ACTION ACT_Build_Ui_Strings:
                      (*
	Send to UI:	First line of Alarms
				First line of Warning
				Stop reason
*)
//PackTag.hevsPackAlarm_UI.uiTextAlarmOne := 'Complete with first Alarm';
BuildUiString := DINT_TO_STRING(PackTag.Admin.Alarm[0].ID);
BuildUiString := CONCAT(BuildUiString, ' ');
BuildUiString := CONCAT(BuildUiString, PackTag.Admin.Alarm[0].Message);
BuildUiString := CONCAT(BuildUiString, ' ');
BuildUiString := CONCAT(BuildUiString, DINT_TO_STRING(PackTag.Admin.Alarm[0].Category));
BuildUiString := CONCAT(BuildUiString, ' ');
BuildUiString := CONCAT(BuildUiString, DT_TO_STRING(PackTag.Admin.Alarm[0].DateTime));
PackTag.hevsPackAlarm_UI.uiTextAlarmOne := BuildUiString; 


BuildUiString := DINT_TO_STRING(PackTag.Admin.Warning[0].ID);
BuildUiString := CONCAT(BuildUiString, ' ');
BuildUiString := CONCAT(BuildUiString, PackTag.Admin.Warning[0].Message);
BuildUiString := CONCAT(BuildUiString, ' ');
BuildUiString := CONCAT(BuildUiString, DINT_TO_STRING(PackTag.Admin.Warning[0].Category));
BuildUiString := CONCAT(BuildUiString, ' ');
BuildUiString := CONCAT(BuildUiString, DT_TO_STRING(PackTag.Admin.Warning[0].DateTime));
PackTag.hevsPackAlarm_UI.uiTextWarningOne := BuildUiString;

BuildUiString := DINT_TO_STRING(PackTag.Admin.StopReason.ID);
BuildUiString := CONCAT(BuildUiString, ' ');
BuildUiString := CONCAT(BuildUiString, PackTag.Admin.StopReason.Message);
BuildUiString := CONCAT(BuildUiString, ' ');
BuildUiString := CONCAT(BuildUiString, DINT_TO_STRING(PackTag.Admin.StopReason.Category));
BuildUiString := CONCAT(BuildUiString, ' ');
BuildUiString := CONCAT(BuildUiString, DT_TO_STRING(PackTag.Admin.StopReason.DateTime));
PackTag.hevsPackAlarm_UI.uiTextStopReason := BuildUiString;


                    
END_ACTION
END_PROGRAM

(* www.hevs.ch Institut Systemes Industriels Project: HEVS Pack 2022 Author: Cedric Lenoir Date: 2024 August 30 This Function Block compute time statistics *)
FUNCTION_BLOCK FB_PackStatistic
  VAR_INPUT
    Enable : BOOL;
  END_VAR
  VAR_IN_OUT
    plcCurrentTime_s : UDINT;  (* E.g from PackTag.hevsPackTime.Local_date_time_seconds *)
    unitCurrentMode : E_PackModes;
    unitCurrentState : E_PackState;
    unitAdmin : HEVS_PackTag_Admin;
  END_VAR
  VAR_OUTPUT
    Active : BOOL;
  END_VAR
  VAR
    trigModeTimeCurrent : R_TRIG;  (* Detext State / Mode change *)
    trigStateTimeCurrent : R_TRIG;
    memCurrentMode : E_PackModes := E_PackModes.Invalid;
    memCurrentState : E_PackState := E_PackState.eUndefined;
    timeModeAtTrigger_s : UDINT;  (* Start time at trigger to compute current *)
    timeStateAtTrigger_s : UDINT;
    bProgramStarted : BOOL;
    timeProgramStarted_s : UDINT;
    getMemCumTimeMode : DINT;  (* Get Time In CumulativeTime for Mode and or state *)
    getMemCumTimeModeState : DINT;
  END_VAR

                  IF Enable THEN
	trigModeTimeCurrent(clk := (unitCurrentMode <> memCurrentMode));
	trigStateTimeCurrent(clk := (unitCurrentState <> memCurrentState));
	
	IF trigModeTimeCurrent.Q THEN
		timeModeAtTrigger_s := plcCurrentTime_s;
		memCurrentMode := unitCurrentMode;
		// Get Stored value to compute new cummulative time.
		getMemCumTimeMode := unitAdmin.CumulativeTime[0].ModeStateTimes[unitCurrentMode].Mode;
	END_IF
	
	IF trigStateTimeCurrent.Q THEN
		timeStateAtTrigger_s := plcCurrentTime_s;
		memCurrentState := unitCurrentState;
	END_IF
	
	// If mode or state changed
	IF trigModeTimeCurrent.Q  OR
	   trigStateTimeCurrent.Q THEN
	   getMemCumTimeModeState := unitAdmin.CumulativeTime[0].ModeStateTimes[unitCurrentMode].State[memCurrentState];
	END_IF
	
	IF NOT bProgramStarted THEN
		bProgramStarted := TRUE;
		timeProgramStarted_s := plcCurrentTime_s;
	END_IF
	
	unitAdmin.ModeTimeCurrent := UDINT_TO_DINT(plcCurrentTime_s - timeModeAtTrigger_s);
	
	unitAdmin.StateTimeCurrent := UDINT_TO_DINT(plcCurrentTime_s - timeStateAtTrigger_s);
	
	// Default for [*] time from start program
	// No retain, that is number of Sec since last restart.
	unitAdmin.CumulativeTime[0].AccTimeSinceReset := UDINT_TO_DINT(plcCurrentTime_s - timeProgramStarted_s);
	
	// Minimum protection in case of unitCurrentMode exceed 
	//	HEVS_PackTag_GVL.C_MAXMODSTATESTIMES
	IF unitCurrentMode <= HEVS_PackTag_GVL.C_MAXMODSTATESTIMES THEN
		// getMemCumTimeMode is set only at trigger change mode
		unitAdmin.CumulativeTime[0].ModeStateTimes[unitCurrentMode].Mode := getMemCumTimeMode + unitAdmin.ModeTimeCurrent;
	END_IF
	
	// Minimum protection in case of unitCurrentMode exceed 
	//	HEVS_PackTag_GVL.C_MAXMODSTATESTIMES
	// 	HEVS_PackTag_GVL.C_MAXSTATES
	IF unitCurrentMode <= HEVS_PackTag_GVL.C_MAXMODSTATESTIMES AND
	   unitCurrentState <= HEVS_PackTag_GVL.C_MAXSTATES        THEN
		// getMemCumTimeModeState is set only at trigger change of mode OR state 
		unitAdmin.CumulativeTime[0].ModeStateTimes[unitCurrentMode].State[unitCurrentState] := getMemCumTimeModeState +  unitAdmin.StateTimeCurrent;
	END_IF
	
	Active	:= FALSE;
ELSE
	
	Active	:= TRUE;
END_IF




                
END_FUNCTION_BLOCK

(* www.hevs.ch Institut Systemes Industriels Project: HEVS Pack 2022 Author: Cedric Lenoir Date: 2024 August 06 Summary: Used to test and simulate first version of PackMaster Does nothing in Waitstates Wait 2.5 secoond before to return SC in *)
FUNCTION_BLOCK FB_ModuleAxis
  VAR_INPUT
    cornerOne : LREAL;
    cornerTwo : LREAL;
    resetSafePosition : LREAL;
    stSetParam : ST_SetMotionParam;
  END_VAR
  VAR_IN_OUT
    axisRef : MB_AXISIF_REF;
    Status_StateCurrent : DINT;  (* has to take the PackTag Status.StateCurrent *)
  END_VAR
  VAR
    stateLastCycie : E_PackState := E_PackState.eUndefined;  (* Store last cycle at the en of FB call to detect and state change Used to force minimum of one testSC.In = 0 and reset SC once between each SC *)
    actualState : E_PackState := E_PackState.eAborted;
    init : BOOL;
    testSC : TON;
    setSC : BOOL;  (* This Flag is used as result on SC State complete. *)
    stActing : ST_Acting;
    mcReadActualPos : MC_ReadActualPosition;  (* List of Function Blocks *)
    mcReadStatus : MC_ReadStatus;
    mcPower : MC_Power;
    mcMoveAbs : MC_MoveAbsolute;
    mcStop : MC_Stop := (Deceleration := 1);
    mcReset : MC_Reset;
    axisAborting : E_AxisAborting;  (* List of enum for internal states of axes *)
    axisClearing : E_AxisClearing;
    axisResetting : E_AxisResetting;  (* Go to safe position *)
    axisStarting : E_AxisStarting;  (* Go to firs corner *)
    axisStopping : E_AxisStopping;
    axisExecute : E_AxisExecute;
  END_VAR

                  IF NOT init THEN
    init := TRUE;
END_IF

actualState := Status_StateCurrent;

// State machine is implicit because transitions are not set by this FB
// That is: a CASE OF does not have place here

// Eacn State is called via and ACTion with 
//	Condition of state
//	Reset of internal state machine when not used
//	That's why, ACTion MUST not be called in a CASE..OF
//  Order of ACTion is not important, because only one should be executed 
//  In any state
// 
//	IF actualState = E_PackState.eUnsuspending THEN
	// Set to TRUE if no action requested
//	stActing.Unsuspending_SC := TRUE;
//	END_IF

ACT_Aborting();
ACT_Clearing();
ACT_Completing();
ACT_Execute();
ACT_Holding();
ACT_Resetting();
ACT_Starting();
ACT_Stopping();
ACT_Suspending();
ACT_Unholding();
ACT_Unsuspending();

(**********************************************************************************************************************
	Axis
**********************************************************************************************************************)
mcReadStatus(Axis := axisRef,
		     Enable := TRUE);

mcReadActualPos(Axis := axisRef,
                Enable := TRUE);

mcPower(Axis := axisRef,
		Enable := NOT (actualState = E_PackState.eAborted) 		  AND
 				  // In aborting, do not disable while stopping
				  NOT ((actualState = E_PackState.eAborting) AND
                       NOT (axisAborting = E_AxisAborting.eStopping)) AND
				  // E_AxisClearing.eErrorStop should be possible
				  // if actualState = E_PackState.eClearing
				  NOT (axisClearing = E_AxisClearing.eErrorStop));

mcStop(Axis := axisRef,
	   // Stop in case of Stopping
	   // Stop in case of Aborting (before to Disable
	   Deceleration := stSetParam.rDeceleration_mm_s2,	   		
       Execute := (axisStopping = E_AxisStopping.eStopping) OR
                  (axisAborting = E_AxisAborting.eStopping));

mcReset(Axis := axisRef,
        Execute := (axisClearing = E_AxisClearing.eErrorStop) OR
                    axisAborting = E_AxisAborting.eErrorStop);

mcMoveAbs(Axis := axisRef,
          Velocity := stSetParam.rVeloctiy_mm_s,
          Acceleration := stSetParam.rAcceleration_mm_s2,
          Deceleration := stSetParam.rDeceleration_mm_s2,
          Jerk := stSetParam.rJerk_mm_s3); 
		  
mcMoveAbs.Execute := (axisExecute = E_AxisExecute.eSetMoveOne)     OR
                     (axisExecute = E_AxisExecute.eSetMoveTwo)     OR
					 (axisResetting = E_AxisResetting.eMotionInit) OR
					 (axisStarting = E_AxisStarting.eMotionStarting);
(*
	Manage State Complete at the end of the Function Block
*)
			
// For test of State Machine, we use a timer.
// Its allow to have some time to visualise it
// We should remove this timer in production version
testSC(IN := stActing.Clearing_SC 		OR
             stActing.Starting_SC      	OR
             stActing.Execute_SC       	OR
             stActing.Stopping_SC      	OR
             stActing.Aborting_SC      	OR
             stActing.Holding_SC       	OR
             stActing.Unholding_SC     	OR
             stActing.Suspending_SC		OR
             stActing.Unsuspending_SC	OR
             stActing.Resetting_SC     	OR
             stActing.Completing_SC,
        PT := T#2500MS); 

// State Complete if setSC is TRUE,
setSC := testSC.Q AND (stateLastCycie = actualState);

// This Statement MUST be written AFTER evaluation of setSC
stateLastCycie := actualState;



                

ACTION ACT_Clearing:
                      (*
	Manage Clearing
*)

// actualState is actual state of Unit from:
//	PackTag.Status.StateCurrent
//
// Wait for : stActing.Clearing_SC : TRUE
// While not all units SC, actualState remains in eClearing.
//
// From PLCopen Motion, the axis at start could be
// Standstill	--> Enabled
// Disabled		--> Need an enable for SC
// ErrorStop	--> Need a reset befoire to be enabled
IF actualState = E_PackState.eClearing THEN
	CASE axisClearing OF
		E_AxisClearing.eIdle :
			IF mcReadStatus.Standstill THEN
				axisClearing := E_AxisClearing.eEnabled;
			ELSIF mcReadStatus.ErrorStop THEN
				axisClearing := E_AxisClearing.eErrorStop;
			ELSE
				axisClearing := E_AxisClearing.eDisabled;
			END_IF
		
		E_AxisClearing.eErrorStop :
			IF mcReadStatus.Standstill THEN
				axisClearing := E_AxisClearing.eEnabled;
			ELSE
				axisClearing := E_AxisClearing.eDisabled;
			END_IF
		
		E_AxisClearing.eDisabled  :
			IF mcReadStatus.Standstill THEN
				axisClearing := E_AxisClearing.eEnabled;
			ELSIF mcReadStatus.ErrorStop THEN
				axisClearing := E_AxisClearing.eErrorStop;
			END_IF
		
		E_AxisClearing.eEnabled   :
			IF mcReadStatus.ErrorStop THEN
				axisClearing := E_AxisClearing.eErrorStop;
			END_IF
	END_CASE
	stActing.Clearing_SC := (axisClearing = E_AxisClearing.eEnabled);
ELSE
	stActing.Clearing_SC := FALSE;
	axisClearing := E_AxisClearing.eIdle; 
END_IF

                    
END_ACTION

ACTION ACT_Starting:
                      (*
	Manage Starting
*)
IF actualState = E_PackState.eStarting THEN
	CASE axisStarting OF
		E_AxisStarting.eIdle :
			axisStarting := E_AxisStarting.eMotionStarting;
			
		E_AxisStarting.eMotionStarting :
			IF mcMoveAbs.Done THEN
				axisStarting := E_AxisStarting.eMotionStartingDone;
			END_IF;
	
		E_AxisStarting.eMotionStartingDone :
			;
	
	END_CASE
	stActing.Starting_SC := (axisStarting = E_AxisStarting.eMotionStartingDone);
ELSE
	stActing.Starting_SC := FALSE;
	axisStarting := E_AxisStarting.eIdle;
END_IF
                    
END_ACTION

ACTION ACT_Execute:
                      (*
	Manage Execute
*)
IF actualState = E_PackState.eExecute THEN
	CASE axisExecute OF
		E_AxisExecute.eIdle :
			axisExecute := E_AxisExecute.eSetMoveOne;
			mcMoveAbs.Position := cornerOne;
			
		E_AxisExecute.eSetMoveOne :
			IF mcMoveAbs.Done THEN
				axisExecute := E_AxisExecute.eMoveOneDone;
			END_IF;
	
		E_AxisExecute.eMoveOneDone :
			mcMoveAbs.Position := cornerTwo;
			axisExecute := E_AxisExecute.eSetMoveTwo;

		E_AxisExecute.eSetMoveTwo :
			IF mcMoveAbs.Done THEN
				axisExecute := E_AxisExecute.eMoveTwoDone;
			END_IF;
	
		E_AxisExecute.eMoveTwoDone :
			mcMoveAbs.Position := cornerOne;
			axisExecute := E_AxisExecute.eSetMoveOne;
	
	END_CASE
ELSE
	axisExecute := E_AxisExecute.eIdle;
END_IF

                    
END_ACTION

ACTION ACT_Stopping:
                      (*
	Manage Stopping
*)
IF actualState = E_PackState.eStopping THEN
	CASE axisStopping OF
		E_AxisStopping.eIdle :
			IF mcReadStatus.Disabled THEN
				axisStopping := E_AxisStopping.eStopped;
			ELSIF mcReadStatus.ErrorStop THEN
				axisStopping := E_AxisStopping.eStopped;
			ELSIF mcReadStatus.Standstill THEN
				axisStopping := E_AxisStopping.eStopped;
			ELSE 
				axisStopping := E_AxisStopping.eStopping;
			END_IF
		E_AxisStopping.eStopping :
			IF mcReadStatus.Disabled THEN
				axisStopping := E_AxisStopping.eStopped;
			ELSIF mcReadStatus.ErrorStop THEN
				axisStopping := E_AxisStopping.eStopped;
			ELSIF mcReadStatus.Standstill THEN
				axisStopping := E_AxisStopping.eStopped;
			END_IF;
	
		E_AxisStopping.eStopped :
			;
	
	END_CASE
	stActing.Stopping_SC := (axisStopping = E_AxisStopping.eStopped);
ELSE
	stActing.Stopping_SC := FALSE;
	axisStopping := E_AxisStopping.eIdle;
END_IF
                    
END_ACTION

ACTION ACT_Aborting:
                      (*
	Manage Aborting
*)
IF actualState = E_PackState.eAborting THEN
	CASE axisAborting OF
		E_AxisAborting.eIdle :
			IF mcReadStatus.Disabled THEN
				axisAborting := E_AxisAborting.eDisabled;
			ELSIF mcReadStatus.ErrorStop THEN
				axisAborting := E_AxisAborting.eErrorStop;
			ELSIF mcReadStatus.Standstill THEN
				axisAborting := E_AxisAborting.eStandstill;
			ELSE 
				axisAborting := E_AxisAborting.eStopping;
			END_IF
		E_AxisAborting.eStopping :
			IF mcReadStatus.Disabled THEN
				axisAborting := E_AxisAborting.eDisabled;
			ELSIF mcReadStatus.ErrorStop THEN
				axisAborting := E_AxisAborting.eErrorStop;
			ELSIF mcReadStatus.Standstill THEN
				axisAborting := E_AxisAborting.eStandstill;
			END_IF;
	
		E_AxisAborting.eStandstill :
			IF mcReadStatus.Disabled THEN
				axisAborting := E_AxisAborting.eDisabled;
			ELSIF mcReadStatus.ErrorStop THEN
				axisAborting := E_AxisAborting.eErrorStop;
			END_IF;;
	
		E_AxisAborting.eErrorStop :
			IF mcReadStatus.Disabled THEN
				axisAborting := E_AxisAborting.eDisabled;
			ELSIF mcReadStatus.Standstill THEN
				axisAborting := E_AxisAborting.eStandstill;
			END_IF;;
	
		E_AxisAborting.eDisabled :
//			IF mcReadStatus.ErrorStop THEN
//				axisAborting := E_AxisAborting.eErrorStop;
//			END_IF		
			;
	END_CASE
	stActing.Aborting_SC := (axisAborting = E_AxisAborting.eDisabled);
ELSE
	stActing.Aborting_SC := FALSE;
	axisAborting := E_AxisAborting.eIdle;
END_IF

                    
END_ACTION

ACTION ACT_Holding:
                      (*
	Manage Holding
*)
IF actualState = E_PackState.eHolding THEN
	// Set to TRUE if no action requested
	stActing.Holding_SC := TRUE;
END_IF

                    
END_ACTION

ACTION ACT_Unholding:
                      (*
	Manage Unholding
*)
IF actualState = E_PackState.eUnholding THEN
	// Set to TRUE if no action requested
	stActing.Unholding_SC := TRUE;
END_IF

                    
END_ACTION

ACTION ACT_Suspending:
                      (*
	Manage Suspending
*)
IF actualState = E_PackState.eSuspending THEN
	// Set to TRUE if no action requested
	stActing.Suspending_SC := TRUE;
END_IF
                    
END_ACTION

ACTION ACT_Unsuspending:
                      (*
	Manage Unsuspending
*)
IF actualState = E_PackState.eUnsuspending THEN
	// Set to TRUE if no action requested
	stActing.Unsuspending_SC := TRUE;
END_IF

                    
END_ACTION

ACTION ACT_Resetting:
                      (*
	Manage Resetting
*)
IF actualState = E_PackState.eResetting THEN
	CASE axisResetting OF
		E_AxisResetting.eIdle :
		    mcMoveAbs.Position := resetSafePosition;
			axisResetting := E_AxisResetting.eMotionInit;
			
		E_AxisResetting.eMotionInit :
			IF mcMoveAbs.Done THEN
				axisResetting := E_AxisResetting.eMotionInitDone;
			END_IF;
	
		E_AxisResetting.eMotionInitDone :
			;
	
	END_CASE
	stActing.Resetting_SC := (axisResetting = E_AxisResetting.eMotionInitDone);
ELSE
	stActing.Resetting_SC := FALSE;
	axisResetting := E_AxisResetting.eIdle;
END_IF
                    
END_ACTION

ACTION ACT_Completing:
                      (*
	Manage Completing
*)
IF actualState = E_PackState.eCompleting THEN
	// Set to TRUE if no action requested
	stActing.Completing_SC := TRUE;
END_IF

                    
END_ACTION

PROPERTY SC : BOOL
GET
                          SC := setSC;
                        
END_GET
END_PROPERTY
END_FUNCTION_BLOCK

(* www.hevs.ch Institut Systemes Industriels Project: Projet No: PW Move Absolute Author: Cedric Lenoir Date: 2024 April 02 Summary: Template of a program using PLCopen on partial Pack State Use a Cyclic Setpoint for motion in Pack Execute. *)
PROGRAM PRG_Process
  VAR
    uliCount : ULINT;  (* ********************************************************************************************************************* YOUR VARIABLES HERE ********************************************************************************************************************* *)
    bInitDone : BOOL;
    stSetParam : ST_SetMotionParam := (rVeloctiy_mm_s := 200, rAcceleration_mm_s2 := 1000, rDeceleration_mm_s2 := 1000, rJerk_mm_s3 := 10000);  (* Pack Partial state machine *)
    stCornerX : ST_Corner := (cornerOne := 20, cornerTwo := 10);
    stCornerY : ST_Corner := (cornerOne := 30, cornerTwo := 13);
    stCornerZ : ST_Corner := (cornerOne := 40, cornerTwo := 14);
    fbModuleAxis_X : FB_ModuleAxis;
    fbModuleAxis_Y : FB_ModuleAxis;
    fbModuleAxis_Z : FB_ModuleAxis;
  END_VAR

                  
fbModuleAxis_X(axisRef := GVL_AxisDefines.X_Axis,
			  resetSafePosition := 10,
			  cornerOne := stCornerX.cornerOne,
			  cornerTwo := stCornerX.cornerTwo,
			  stSetParam := stSetParam,
			  Status_StateCurrent := PackTag.Status.StateCurrent);
			  
fbModuleAxis_Y(axisRef := GVL_AxisDefines.Y_Axis,
			  resetSafePosition := 11,
			  cornerOne := stCornerY.cornerOne,
			  cornerTwo := stCornerY.cornerTwo,
			  stSetParam := stSetParam,
			  Status_StateCurrent := PackTag.Status.StateCurrent);

fbModuleAxis_Z(axisRef := GVL_AxisDefines.Z_Axis,
			  resetSafePosition := 12,
			  cornerOne := stCornerZ.cornerOne,
			  cornerTwo := stCornerZ.cornerTwo,	
			  stSetParam := stSetParam,			  
			  Status_StateCurrent := PackTag.Status.StateCurrent);

                
END_PROGRAM

CONFIGURATION Application
  RESOURCE Application ON PLC
    {attribute 'qualified_only'}
    VAR_GLOBAL CONSTANT  (* HEVS_PackTag_GVL - List of PackTags based on ISA–TR88.00.02-2022 www.hevs.ch Institut Systemes Industriels / Power & Control Project: Automation Box CtrlX S3 Author: Romain Ferrari & Cedric Lenoir Date: 2024 July 31 !!!!!! The value of these constants have to be set by the user depending on the system it is implemented on. !!!!!!\\ *)
      C_MAXSTATES : INT := 17;  (* Max State number. 0 is invalid *)
      C_COMMAND_MAXREALPARAMS : INT := 8;
      C_COMMAND_MAXSTRINGPARAMS : INT := 2;  (* / *)
      C_COMMAND_MAXLREALPARAMS : INT := 8;  (* Used in one of the main PackTag branch of the HEVS_PackTag_V30 : Command *)
      C_COMMAND_MAXDINTPARAMS : INT := 8;
      C_COMMAND_MAXRECIPE : INT := 8;
      C_STATUS_MAXREALPARAMS : INT := 8;  (* / *)
      C_STATUS_MAXSTRINGPARAMS : INT := 2;  (* / *)
      C_STATUS_MAXLREALPARAMS : INT := 8;
      C_STATUS_MAXDINTPARAMS : INT := 8;  (* Used in one of the main PackTag branch of the HEVS_PackTag_V30 : Status *)
      C_STATUS_MAXRECIPE : INT := 8;
      C_STATUS_MAXSTACKLIGHT : INT := 8;
      C_ADMIN_MAXREALPARAMS : INT := 8;  (* / *)
      C_ADMIN_MAXSTRINGPARAMS : INT := 2;  (* / *)
      C_ADMIN_MAXLREALPARAMS : INT := 8;
      C_ADMIN_MAXDINTPARAMS : INT := 8;
      C_ADMIN_MAXALARMS : INT := 20;
      C_ADMIN_MAXHISTORYALARMS : INT := 20;
      C_ADMIN_MAXWARNINGS : INT := 20;
      C_ADMIN_MAXCUMULATIVETIMES : INT := 3;  (* Minimum is 0 for [0], Arbitrarily initialized to 3 *)
      C_ADMIN_MAXPRODUCTDATA : INT := 11;
      C_ADMIN_MAXDISABLEDSTATES : INT := 8;
      C_ADMIN_MAXMODESTRANSITION : INT := 8;  (* is absolutely limited by C_ADMIN_MAXMODESTRANSITIONPACK *)
      C_ADMIN_MAXMODESTRANSITIONPACK : INT := 31;  (* as Pack used DWORD and 0 is reserved, max is limited to 31 *)
      C_MAXMODSTATESTIMES : INT := 8;
      C_MAXREALVARIABLES : INT := 8;
      C_MAXSTRINGVARIABLES : INT := 8;
      C_MAXLREALVARIABLES : INT := 8;
      C_MAXDINTVARIABLES : INT := 8;  (* Used in lower branches of the HEVS_PackTag_V30 *)
      C_MAXREALINGREDIENTS : INT := 8;
      C_MAXSTRINGINGREDIENTS : INT := 8;
      C_MAXLREALINGREDIENTS : INT := 8;
      C_MAXDINTINGREDIENTS : INT := 8;
      hevs_min_packtag_v2022 : HEVS_Min_PackTag_V2022;
    END_VAR
    {attribute 'qualified_only'}
    VAR_GLOBAL  (* PackTag - www.hevs.ch Institut Systemes Industriels Project: HEVS Pack 2022 Author: Cedric Lenoir Date: 2024 August 29 Base GVL for HEVS Pack Tag File name should be PackTag *)
      Command : HEVS_PackTag_Command;
      Status : HEVS_PackTag_Status;
      Admin : HEVS_PackTag_Admin;
      hevsPackTime : HEVS_Time;  (* HEVS Time, needed for Alarms and Time in Pack Computed with PRG_GetTime_CtrlX or PRG_GetTime_TwinCAT or Your own system *)
      hevsUI : HEVS_PackTag_UI;  (* Help for interface and diagnostic HEVS Pack could be used without this Struct. Can be used with fbCmdBoolInterface Can be used with fbGetActualBoolState *)
      hevsPackAlarm_UI : HEVS_PackAlarm_UI;  (* Help for interface and diagnostic HEVS Pack could be used without this Struct. Can be used with program PRG_TestAlarm *)
    END_VAR
    {attribute 'qualified_only'}
    VAR_GLOBAL  (* GVL_Node - Some GVL to test var with NodeRED. Source: www.hevs.ch Author: Cedric Lenoir Date: 22 August 2024 *)
      readREAL : REAL;
      readDINT : DINT;
      readBOOL : BOOL;
      readString : STRING;
      writeREAL : REAL;
      writeDINT : DINT;
      writeBOOL : BOOL;
    END_VAR
    {attribute 'qualified_only'}
    VAR_GLOBAL  (* GVL_AxisDefines *)
      X_Axis : MB_AXISIF_REF := (AxisName := 'Axis_X', AxisNo := 1);
      Y_Axis : MB_AXISIF_REF := (AxisName := 'Axis_Y', AxisNo := 2);
      Z_Axis : MB_AXISIF_REF := (AxisName := 'Axis_Z', AxisNo := 3);
    END_VAR
    TASK MainTask(INTERVAL := T#40ms, PRIORITY := 30);
    PROGRAM PLC_PACK WITH MainTask : PLC_PACK;
    PROGRAM PRG_TestAlarm WITH MainTask : PRG_TestAlarm;
    PROGRAM PRG_Sandbox WITH MainTask : PRG_Sandbox;
    PROGRAM PRG_GetTime_CtrlX WITH MainTask : PRG_GetTime_CtrlX;
    PROGRAM PRG_Process WITH MainTask : PRG_Process;
  END_RESOURCE
END_CONFIGURATION
